(* CoDeSys 2.3 export: BYTE_TO_VAR.EXP *)

(* POU FUNv1/BYTE_TO_VAR, ST *)
FUNCTION BYTE_TO_VAR : VarST
VAR_IN_OUT
    in: BYTE;
END_VAR
VAR
END_VAR
BYTE_TO_VAR.pby   := ADR(in);
BYTE_TO_VAR.type_ := BYTE_;
END_FUNCTION
